// TIA Portal project "Profibus_Edge_HowTo" (V17)

(* hardware
DEVICE "S7-300/ET200M station_1"  S7-300 station
   slot 0: "Rail_0"  Rail  6ES7 390-1***0-0AA0
   slot 2: "PLC_1"  CPU 315-2 DP  6ES7 315-2AG10-0AB0  V2.6
      slot 0: "MPI interface_1"  X1
      slot 1: "DP interface_1"  X2
*)

// ===== PLC "PLC_1"  CPU 315-2 DP =====

VAR_GLOBAL   // PLC tag table "Default tag table"
   "Data" AT %I0.0 : Bool;
END_VAR

DATA_BLOCK "ProcessData"   // DB1
{ S7_Optimized_Access := 'FALSE' }
VERSION : 0.1
   VAR
      stringValue : String := 'Connection alive';
      intValue : Int := 10;
      realValue : Real := 3.3;
      boolValue : Bool;
      intValueEdge2Plc : Int;
   END_VAR
BEGIN
END_DATA_BLOCK

FUNCTION "GenerateValues" : Void   // FC1, SCL
{ S7_Optimized_Access := 'FALSE' }
VERSION : 0.1
BEGIN
   IF "ProcessData".intValue < 100 THEN
       "ProcessData".intValue := "ProcessData".intValue + 1;
       "ProcessData".realValue := "ProcessData".realValue + 2;
       "ProcessData".boolValue := NOT "ProcessData".boolValue;
       "ProcessData".stringValue := CONCAT(IN1 := 'Current int value = ',IN2 := INT_TO_STRING ("ProcessData".intValue));
   ELSE
       "ProcessData".intValue := 0;
       "ProcessData".realValue := 0.3;
   END_IF;
END_FUNCTION

ORGANIZATION_BLOCK "CYC_INT"   // OB35, LAD
TITLE = "Cyclic Interrupt"
{ S7_Optimized_Access := 'FALSE' }
VERSION : 0.1
   VAR_TEMP
      OB35_EV_CLASS : Byte;   // Bits 0-3 = 1 (Coming event), Bits 4-7 = 1 (Event class 1)
      OB35_STRT_INF : Byte;   // 16#36 (OB 35 has started)
      OB35_PRIORITY : Byte;   // Priority of OB Execution
      OB35_OB_NUMBR : Byte;   // 35 (Organization block 35, OB35)
      OB35_RESERVED_1 : Byte;   // Reserved for system
      OB35_RESERVED_2 : Byte;   // Reserved for system
      OB35_PHASE_OFFSET : Word;   // Phase offset (msec)
      OB35_RESERVED_3 : Int;   // Reserved for system
      OB35_EXC_FREQ : Int;   // Frequency of execution (msec)
      OB35_DATE_TIME : Date_And_Time;   // Date and time OB35 started
   END_VAR
BEGIN

REGION Network 1
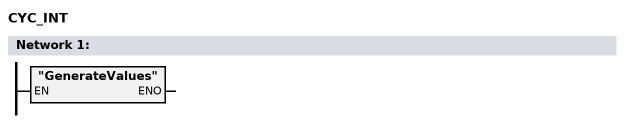
   RUNG wire#powerrail
      "GenerateValues"()
   END_RUNG
   // the same network as SCL:
   "GenerateValues"();
END_REGION
END_ORGANIZATION_BLOCK

(* ===== HMI "HMI_RT_1" =====
system functions are stored by id; their names below are inferred from use

ScreenModuleEditorView "ValueStepperInt_Vertical2" 640x480
   IOField "ioValue" at 0,48 size 80x40; FormatPattern 999999
      ProcessValue <- "value"
   Button "btnIncrease" at 0,0 size 80x40; TextOff 'Text'
      on Click: function_dd21b452("value", "delta")
   Button "btnDecrease" at 0,96 size 80x40; TextOff 'Text'
      on Click: function_b9b71300("value", "delta")
*)